FUNCTION_BLOCK FB_DriveWinch IMPLEMENTS IF_DriveVariableVel
VAR_INPUT
	bLimitTop, bLimitBottom : BOOL;						(* limit switches *)
END_VAR
VAR_OUTPUT
	bDriveEnable : BOOL;								(* Lift drive enable *)
	nDriveVelocity : INT;								(* Lift drive velocity *)
END_VAR
VAR

END_VAR

PROPERTY bBOTTOM : BOOL
GET
bBOTTOM := bLimitBottom;
END_GET
END_PROPERTY

PROPERTY bTOP : BOOL
GET
bTOP := bLimitTop;
END_GET
END_PROPERTY

METHOD lifEnable
bDriveEnable := TRUE;
END_METHOD

METHOD liftDisable
bDriveEnable := FALSE;
END_METHOD

METHOD moveVarSpeed
VAR_INPUT
	nSetVelocity : INT;						(* velocity setpoint *)
	eDirection : LiftMovingDirection;		(* moving direction: up or down *)
END_VAR
bDriveEnable := TRUE;

IF eDirection > 0 THEN
	eDirection := LiftMovingDirection.up;
END_IF
IF eDirection < 0 THEN
	eDirection := LiftMovingDirection.down; 
END_IF

nSetVelocity := ABS(nSetVelocity);
IF nSetVelocity > 10000 THEN
	nSetVelocity := 10000;
END_IF

IF bLimitTop AND eDirection = LiftMovingDirection.up THEN
	stop();
ELSIF bLimitBottom AND eDirection = LiftMovingDirection.down THEN
	stop();
ELSE
	nDriveVelocity := eDirection*nSetVelocity;
END_IF
END_METHOD

METHOD stop
nDriveVelocity := 0;
END_METHOD

END_FUNCTION_BLOCK

(* stored: Version 1.1.0.1, ProductVersion 3.1.4024.6
   POU FB_DriveWinch: Id {ea04fc71-84e4-49f0-8d06-b8ced5385672}, SpecialFunc None
   Property bBOTTOM: Id {93d4f6ee-9753-44db-8f76-44fd23bf93cd}
   Get Get: Id {abf09bdd-7cdc-4cd5-b9eb-6ccebd8d9180}
   Property bTOP: Id {98558438-0e94-43e1-94e4-72dc4d5e85fc}
   Get Get: Id {b99dedea-0e19-48b7-b926-7fbc4ca54f70}
   Method lifEnable: Id {cf793a26-ba8e-4a8b-a436-4f27f77b34a4}
   Method liftDisable: Id {0d15b034-5a60-47da-875a-222ee32c7c20}
   Method moveVarSpeed: Id {c315ae90-2502-42c2-8273-764b750c3ef6}
   Method stop: Id {6cb4507f-0f7d-4fa1-bd5d-3e548eb4cbae} *)
